(****************************************************************
NAME:			FB_Move
DATA:			2017.2.17
VERSION:		1.0.0
DESCRIPTION:	FB_Move
HISTORY:
				2017.2.17		NEW
				2018.1.9		ÐÂÔöBCGapMode
***************************************************************)
FUNCTION_BLOCK FB_Move
VAR_INPUT
	(*È«¾Ö*)
	Mode:DINT;
	PowerState:BOOL;
	CoupleState:DINT;
	(*BCGapMode*)
	BCLeftTopPosition:LREAL;
	BCLeftTopVelocity:LREAL;
	BCRightTopPosition:LREAL;
	BCRightTopVelocity:LREAL;
	BCLeftBottomPosition:LREAL;
	BCLeftBottomVelocity:LREAL;
	BCRightBottomPosition:LREAL;
	BCRightBottomVelocity:LREAL;
	BCGapMove:BOOL;
	BCGapReset:BOOL;
	BCGapMove_2:BOOL;
	BCGapReset_2:BOOL;
	(*GapMode*)
	GapPosition:LREAL;
	GapVelocity:LREAL;
	GapMove:BOOL;
	GapReset:BOOL;
	(*SingleCarrierMode*)
	TopPosition:LREAL;
	TopVelocity:LREAL;
	TopMove:BOOL;
	TopReset:BOOL;
	BottomPosition:LREAL;
	BottomVelocity:LREAL;
	BottomMove:BOOL;
	BottomReset:BOOL;
	(*TaperMode*)
	TaperPosition:LREAL;
	TaperVelocity:LREAL;
	TaperMove:BOOL;
	TaperStop:BOOL;
	TaperReset:BOOL;
	(**DebugMode*)
	LeftTopPosition:LREAL;
	LeftTopVelocity:LREAL;
	LeftTopMove:BOOL;
	LeftTopStop:BOOL;
	LeftTopReset:BOOL;
	RightTopPosition:LREAL;
	RightTopVelocity:LREAL;
	RightTopMove:BOOL;
	RightTopStop:BOOL;
	RightTopReset:BOOL;
	LeftBottomPosition:LREAL;
	LeftBottomVelocity:LREAL;
	LeftBottomMove:BOOL;
	LeftBottomStop:BOOL;
	LeftBottomReset:BOOL;
	RightBottomPosition:LREAL;
	RightBottomVelocity:LREAL;
	RightBottomMove:BOOL;
	RightBottomStop:BOOL;
	RightBottomReset:BOOL;
	PhaseUpperPosition:LREAL;
	PhaseUpperVelocity:LREAL;
	PhaseUpperMove:BOOL;
	PhaseUpperStop:BOOL;
	PhaseUpperReset:BOOL;
	PhaseLowerPosition:LREAL;
	PhaseLowerVelocity:LREAL;
	PhaseLowerMove:BOOL;
	PhaseLowerStop:BOOL;
	PhaseLowerReset:BOOL;
END_VAR
VAR_OUTPUT
	FbID:DINT:=1001;
	GapState:DINT;
	GapBusy:BOOL;
	GapDone:BOOL;
	GapMoving:BOOL;

	BCGapState:DINT;
	BCGapBusy:BOOL;
	BCGapDone:BOOL;

	TopState:DINT;
	TopBusy:BOOL;
	TopDone:BOOL;
	BottomState:DINT;
	BottomBusy:BOOL;
	BottomDone:BOOL;

	TaperState:DINT;
	TaperBusy:BOOL;
	TaperDone:BOOL;

	LeftTopState:DINT;
	LeftTopBusy:BOOL;
	LeftTopDone:BOOL;
	RightTopState:DINT;
	RightTopBusy:BOOL;
	RightTopDone:BOOL;
	LeftBottomState:DINT;
	LeftBottomBusy:BOOL;
	LeftBottomDone:BOOL;
	RightBottomState:DINT;
	RightBottomBusy:BOOL;
	RightBottomDone:BOOL;
	PhaseUpperState:DINT;
	PhaseUpperBusy:BOOL;
	PhaseUpperDone:BOOL;
	PhaseLowerState:DINT;
	PhaseLowerBusy:BOOL;
	PhaseLowerDone:BOOL;

	Error:BOOL;
	ErrorID:DINT;
	
	GapState_2:DINT;
	GapBusy_2:BOOL;
	GapDone_2:BOOL;

	BCGapState_2:DINT;
	BCGapBusy_2:BOOL;
	BCGapDone_2:BOOL;
END_VAR
VAR
	Top_MC_MoveAbsolute: MC_MoveAbsolute;
	Bottom_MC_MoveAbsolute: MC_MoveAbsolute;
	RightTopLin_MC_MoveAbsolute: MC_MoveAbsolute;
	RightBottomLin_MC_MoveAbsolute: MC_MoveAbsolute;
	PhaseUpperLin_MC_MoveAbsolute: MC_MoveAbsolute;
	PhaseLowerLin_MC_MoveAbsolute: MC_MoveAbsolute;
	fb_ton: TON;
	fb_ton1: TON;
	fb_ton2: TON;
	fb_ton_debug_1:TON;
	fb_ton_debug_2:TON;
	fb_ton_debug_3:TON;
	fb_ton_debug_4:TON;
	fb_ton_debug_5:TON;
	fb_ton_debug_6:TON;
	fb_ton_BC:TON;
	fb_ton_BC_2:TON;
END_VAR

IF PowerState=1 THEN
	IF Mode=1 AND CoupleState=1 THEN
		A_GapMove();
	ELSIF Mode=2 AND CoupleState=0 AND TopMove THEN
		A_TopMove();
	ELSIF Mode=2 AND CoupleState=0 AND BottomMove THEN
		A_BottomMove();
	ELSIF Mode=3 AND CoupleState=0 AND TaperMove THEN
		A_TaperMove();
	ELSIF Mode=4 AND CoupleState=0 AND LeftTopMove THEN
		A_LeftTopMove();
	ELSIF Mode=4 AND CoupleState=0 AND RightTopMove THEN
		A_RightTopMove();
	ELSIF Mode=4 AND CoupleState=0 AND LeftBottomMove THEN
		A_LeftBottomMove();
	ELSIF Mode=4 AND CoupleState=0 AND RightBottomMove THEN
		A_RightBottomMove();
	ELSIF Mode=4 AND CoupleState=0 AND PhaseUpperMove THEN
		A_PhaseUpperMove();
	ELSIF Mode=4 AND CoupleState=0 AND PhaseLowerMove THEN
		A_PhaseLowerMove();
	ELSIF Mode=5 AND CoupleState=0 AND BCGapMove THEN
		A_BCGapMove();
	ELSIF Mode=6 AND CoupleState=0 AND BCGapMove_2 THEN
		A_BCGapMove_2();
	END_IF
END_IF

ACTION A_BCGapMove:
IF BCGapMove THEN
	BCGapBusy:=TRUE;
	BCGapDone:=FALSE;
	fb_ton_BC(PT:=t#80s);(*2mm/s max spees,120mmÐÐ³Ì£¬60sÄÚ×ßÍê*)
	(*×îºóÔÙ¼ì²éÒ»±éñîºÏ£¬²¹³¥Ä£Ê½ÏÂ£¬²»ÄÜñîºÏ*)
	IF LeftTopLin.NcToPlc.CoupleState<>0 OR LeftBottomLin.NcToPlc.CoupleState<>0
				OR RightTopLin.NcToPlc.CoupleState<>0 OR RightBottomLin.NcToPlc.CoupleState<>0 THEN
				ErrorID:=1;
				GapState:=-100;
	END_IF
	A_MoveMC();
	IF  LeftTopLin.Status.Moving AND RightTopLin.Status.Moving
				 AND LeftBottomLin.Status.Moving AND RightBottomLin.Status.Moving THEN
		GapMoving:=TRUE;
	ELSE
		GapMoving:=FALSE;
	END_IF
	CASE BCGapState OF
		0:
			IF LeftTopLin.Status.Moving OR RightTopLin.Status.Moving
				 OR LeftBottomLin.Status.Moving OR RightBottomLin.Status.Moving THEN	(*ÖáÕýÔÚÔËÐÐ£¬Ñ­»·¸Ã²½µÈ´ý*)
				BCGapState:=88;
			//ELSIF Top_MC_MoveAbsolute.Error OR Bottom_MC_MoveAbsolute.Error OR
			//		RightTopLin_MC_MoveAbsolute.Error OR RightBottomLin_MC_MoveAbsolute.Error THEN	(*¼ì²éMC Error*)
			//	ErrorID:=2;
			//	BCGapState:=99;
			(*ELSIF ABS(Pos_LeftTopLin-GapPosition/2)<0.002 AND  ABS(Pos_LeftBottomLin-GapPosition)<0.002 THEN	(*Ä¿±êÎ»ÖÃÓëµ±Ç°Î»ÖÃÒ»Ñù£¬²»¶¯*)
				GapState:=88;*)
			ELSIF leftTopLin.Status.NotMoving AND  leftBottomLin.Status.NotMoving
				 AND RightTopLin.Status.NotMoving AND RightBottomLin.Status.NotMoving THEN	(*Öá¶¼´¦ÓÚÍ£Ö¹×´Ì¬Ê±£¬×ªÏÂÒ»²½*)
				BCGapState:=1;
			END_IF
		1:
			Top_MC_MoveAbsolute.Position:=BCLeftTopPosition;
			Top_MC_MoveAbsolute.Velocity:=BCLeftTopVelocity;
			Bottom_MC_MoveAbsolute.Position:=BCLeftBottomPosition;
			Bottom_MC_MoveAbsolute.Velocity:=BCLeftBottomVelocity;
			RightTopLin_MC_MoveAbsolute.Position:=BCRightTopPosition;
			RightTopLin_MC_MoveAbsolute.Velocity:=BCRightTopVelocity;
			RightBottomLin_MC_MoveAbsolute.Position:=BCRightBottomPosition;
			RightBottomLin_MC_MoveAbsolute.Velocity:=BCRightBottomVelocity;
			Top_MC_MoveAbsolute.Execute:=TRUE;
			Bottom_MC_MoveAbsolute.Execute:=TRUE;
			RightTopLin_MC_MoveAbsolute.Execute:=TRUE;
			RightBottomLin_MC_MoveAbsolute.Execute:=TRUE;
			fb_ton_BC.IN:=TRUE;
			BCGapState:=2;
		2:
			IF NOT Top_MC_MoveAbsolute.Done OR NOT  Bottom_MC_MoveAbsolute.Done
					OR NOT RightTopLin_MC_MoveAbsolute.Done OR NOT RightBottomLin_MC_MoveAbsolute.Done THEN		(*ÔË¶¯ÖÐ£¬¼ì²éDoneÐÅºÅ£¬Ã»ÓÐÔòÑ­»·*)
				BCGapState:=2;
			ELSIF Top_MC_MoveAbsolute.Done  AND  Bottom_MC_MoveAbsolute.Done AND RightTopLin_MC_MoveAbsolute.Done AND RightBottomLin_MC_MoveAbsolute.Done THEN		(*ÔË¶¯Íê³É£¬×ªÏÂÒ»²½*)
				BCGapState:=88;
			END_IF
		88:
			BCGapMove:=FALSE;
			BCGapState:=0;
			BCGapBusy:=FALSE;
			BCGapDone:=TRUE;
			Error:=FALSE;
			ErrorID:=0;
			Top_MC_MoveAbsolute.Execute:=FALSE;
			Bottom_MC_MoveAbsolute.Execute:=FALSE;
			RightTopLin_MC_MoveAbsolute.Execute:=FALSE;
			RightBottomLin_MC_MoveAbsolute.Execute:=FALSE;
			fb_ton_BC.IN:=FALSE;
		89:
			BCGapMove:=FALSE;
			BCGapState:=0;
			BCGapBusy:=FALSE;
			BCGapDone:=FALSE;
			Error:=FALSE;
			ErrorID:=0;
			Top_MC_MoveAbsolute.Execute:=FALSE;
			Bottom_MC_MoveAbsolute.Execute:=FALSE;
			RightTopLin_MC_MoveAbsolute.Execute:=FALSE;
			RightBottomLin_MC_MoveAbsolute.Execute:=FALSE;
			fb_ton_BC.IN:=FALSE;
		99:
			BCGapMove:=FALSE;
			BCGapState:=99;
			BCGapBusy:=FALSE;
			BCGapDone:=FALSE;
			Error:=TRUE;
			Top_MC_MoveAbsolute.Execute:=FALSE;
			Bottom_MC_MoveAbsolute.Execute:=FALSE;
			RightTopLin_MC_MoveAbsolute.Execute:=FALSE;
			RightBottomLin_MC_MoveAbsolute.Execute:=FALSE;
			fb_ton_BC.IN:=FALSE;
		-100:
			FB_PlcEmergencyStop();
			BCGapMove:=FALSE;
			BCGapState:=-100;
			BCGapBusy:=FALSE;
			BCGapDone:=FALSE;
			Error:=TRUE;
			Top_MC_MoveAbsolute.Execute:=FALSE;
			Bottom_MC_MoveAbsolute.Execute:=FALSE;
			RightTopLin_MC_MoveAbsolute.Execute:=FALSE;
			RightBottomLin_MC_MoveAbsolute.Execute:=FALSE;
			fb_ton_BC.IN:=FALSE;
	END_CASE

	IF BCGapReset THEN
		BCGapReset:=FALSE;
		BCGapMove:=FALSE;
		BCGapState:=0;
		BCGapBusy:=FALSE;
		BCGapDone:=FALSE;
		Error:=FALSE;
		ErrorID:=0;
		Top_MC_MoveAbsolute.Execute:=FALSE;
		Bottom_MC_MoveAbsolute.Execute:=FALSE;
		RightTopLin_MC_MoveAbsolute.Execute:=FALSE;
		RightBottomLin_MC_MoveAbsolute.Execute:=FALSE;
		fb_ton_BC.IN:=FALSE;
	END_IF
END_IF
END_ACTION

ACTION A_BCGapMove_2:
IF BCGapMove_2 THEN
BCGapBusy_2:=TRUE;
BCGapDone_2:=FALSE;
fb_ton_BC_2(PT:=T#80S);(*2mm/s max spees,120mmÐÐ³Ì£¬60sÄÚ×ßÍê*)
(*×îºóÔÙ¼ì²éÒ»±éñîºÏ£¬²¹³¥Ä£Ê½ÏÂ£¬²»ÄÜñîºÏ*)
IF LeftTopLin.NcToPlc.CoupleState<>0 OR LeftBottomLin.NcToPlc.CoupleState<>0
			OR RightTopLin.NcToPlc.CoupleState<>0 OR RightBottomLin.NcToPlc.CoupleState<>0 THEN
			ErrorID:=1;
			GapState:=-100;
END_IF
A_MoveMC();
CASE BCGapState_2 OF
	0:
		IF LeftTopLin.Status.Moving OR RightTopLin.Status.Moving
			 OR LeftBottomLin.Status.Moving OR RightBottomLin.Status.Moving THEN	(*ÖáÕýÔÚÔËÐÐ£¬Ñ­»·¸Ã²½µÈ´ý*)
			BCGapState_2:=88;
		//ELSIF Top_MC_MoveAbsolute.Error OR Bottom_MC_MoveAbsolute.Error OR
		//		RightTopLin_MC_MoveAbsolute.Error OR RightBottomLin_MC_MoveAbsolute.Error THEN	(*¼ì²éMC Error*)
		//	ErrorID:=2;
		//	BCGapState_2:=99;
		(*ELSIF ABS(Pos_LeftTopLin-GapPosition/2)<0.002 AND  ABS(Pos_LeftBottomLin-GapPosition)<0.002 THEN	(*Ä¿±êÎ»ÖÃÓëµ±Ç°Î»ÖÃÒ»Ñù£¬²»¶¯*)
			GapState:=88;*)
		ELSIF leftTopLin.Status.NotMoving AND  leftBottomLin.Status.NotMoving
			 AND RightTopLin.Status.NotMoving AND RightBottomLin.Status.NotMoving THEN	(*Öá¶¼´¦ÓÚÍ£Ö¹×´Ì¬Ê±£¬×ªÏÂÒ»²½*)
			BCGapState_2:=1;
		END_IF
	1:
		Top_MC_MoveAbsolute.Position:=BCLeftTopPosition;
		Top_MC_MoveAbsolute.Velocity:=BCLeftTopVelocity;
		Bottom_MC_MoveAbsolute.Position:=BCLeftBottomPosition;
		Bottom_MC_MoveAbsolute.Velocity:=BCLeftBottomVelocity;
		RightTopLin_MC_MoveAbsolute.Position:=BCRightTopPosition;
		RightTopLin_MC_MoveAbsolute.Velocity:=BCRightTopVelocity;
		RightBottomLin_MC_MoveAbsolute.Position:=BCRightBottomPosition;
		RightBottomLin_MC_MoveAbsolute.Velocity:=BCRightBottomVelocity;
		Top_MC_MoveAbsolute.Execute:=TRUE;
		Bottom_MC_MoveAbsolute.Execute:=TRUE;
		RightTopLin_MC_MoveAbsolute.Execute:=TRUE;
		RightBottomLin_MC_MoveAbsolute.Execute:=TRUE;
		fb_ton_BC_2.IN:=TRUE;
		BCGapState_2:=2;
	2:
		IF NOT Top_MC_MoveAbsolute.Done OR NOT  Bottom_MC_MoveAbsolute.Done
				OR NOT RightTopLin_MC_MoveAbsolute.Done OR NOT RightBottomLin_MC_MoveAbsolute.Done THEN		(*ÔË¶¯ÖÐ£¬¼ì²éDoneÐÅºÅ£¬Ã»ÓÐÔòÑ­»·*)
			BCGapState_2:=2;
		ELSIF Top_MC_MoveAbsolute.Done  AND  Bottom_MC_MoveAbsolute.Done AND RightTopLin_MC_MoveAbsolute.Done AND RightBottomLin_MC_MoveAbsolute.Done THEN		(*ÔË¶¯Íê³É£¬×ªÏÂÒ»²½*)
			BCGapState_2:=88;
		END_IF
		(*½ÓÊÕµ½stopÐÅºÅÊ±£¬reset×´Ì¬*)
		IF BCGapReset_2 THEN
			BCGapState_2:=89;
		END_IF

	88:
		BCGapMove_2:=FALSE;
		BCGapState_2:=0;
		BCGapBusy_2:=FALSE;
		BCGapDone_2:=TRUE;
		Error:=FALSE;
		ErrorID:=0;
		Top_MC_MoveAbsolute.Execute:=FALSE;
		Bottom_MC_MoveAbsolute.Execute:=FALSE;
		RightTopLin_MC_MoveAbsolute.Execute:=FALSE;
		RightBottomLin_MC_MoveAbsolute.Execute:=FALSE;
		fb_ton_BC_2.IN:=FALSE;
	89:
		BCGapMove_2:=FALSE;
		BCGapState_2:=0;
		BCGapBusy_2:=FALSE;
		BCGapDone_2:=FALSE;
		Error:=FALSE;
		ErrorID:=0;
		Top_MC_MoveAbsolute.Execute:=FALSE;
		Bottom_MC_MoveAbsolute.Execute:=FALSE;
		RightTopLin_MC_MoveAbsolute.Execute:=FALSE;
		RightBottomLin_MC_MoveAbsolute.Execute:=FALSE;
		fb_ton_BC_2.IN:=FALSE;
	99:
		BCGapMove_2:=FALSE;
		BCGapState_2:=99;
		BCGapBusy_2:=FALSE;
		BCGapDone_2:=FALSE;
		Error:=TRUE;
		Top_MC_MoveAbsolute.Execute:=FALSE;
		Bottom_MC_MoveAbsolute.Execute:=FALSE;
		RightTopLin_MC_MoveAbsolute.Execute:=FALSE;
		RightBottomLin_MC_MoveAbsolute.Execute:=FALSE;
		fb_ton_BC_2.IN:=FALSE;
	-100:
		FB_PlcEmergencyStop();
		BCGapMove_2:=FALSE;
		BCGapState_2:=-100;
		BCGapBusy_2:=FALSE;
		BCGapDone_2:=FALSE;
		Error:=TRUE;
		Top_MC_MoveAbsolute.Execute:=FALSE;
		Bottom_MC_MoveAbsolute.Execute:=FALSE;
		RightTopLin_MC_MoveAbsolute.Execute:=FALSE;
		RightBottomLin_MC_MoveAbsolute.Execute:=FALSE;
		fb_ton_BC_2.IN:=FALSE;
END_CASE
END_IF
END_ACTION

ACTION A_BottomMove:
IF BottomMove THEN
BottomBusy:=TRUE;
BottomDone:=FALSE;
fb_ton2(PT:=t#80s);(*2mm/s max spees,120mmÐÐ³Ì£¬60sÄÚ×ßÍê*)
A_MoveMC();
CASE BottomState OF

	0:
		IF LeftTopLin.Status.Moving OR RightTopLin.Status.Moving
			 OR LeftBottomLin.Status.Moving OR RightBottomLin.Status.Moving THEN	(*ÖáÕýÔÚÔËÐÐ£¬Ñ­»·¸Ã²½µÈ´ý*)
			TopState:=88;
		//ELSIF  Bottom_MC_MoveAbsolute.Error OR RightBottomLin_MC_MoveAbsolute.Error THEN		(*¼ì²éMC Error*)
		//	ErrorID:=2;
		//	BottomState:=99;
		ELSIF leftTopLin.Status.NotMoving AND  leftBottomLin.Status.NotMoving
			 AND RightTopLin.Status.NotMoving AND RightBottomLin.Status.NotMoving THEN	(*Öá¶¼´¦ÓÚÍ£Ö¹×´Ì¬Ê±£¬×ªÏÂÒ»²½*)
			BottomState:=1;
		END_IF
	1:
		Bottom_MC_MoveAbsolute.Position:=BottomPosition;
		Bottom_MC_MoveAbsolute.Velocity:=BottomVelocity;
		Bottom_MC_MoveAbsolute.Execute:=TRUE;
		RightBottomLin_MC_MoveAbsolute.Position:=BottomPosition;
		RightBottomLin_MC_MoveAbsolute.Velocity:=BottomVelocity;
		RightBottomLin_MC_MoveAbsolute.Execute:=TRUE;
		fb_ton2.IN:=TRUE;
		BottomState:=2;
	2:
		IF leftTopLin.Status.Moving OR RightTopLin.Status.Moving THEN	(*ÉÏÁº¶¯,ESTOP*)
			ErrorID:=3;
			BottomState:=-100;
		ELSIF  (LeftBottomLin.Status.Moving AND  RightBottomLin.Status.NotMoving)
				OR (RightBottomLin.Status.Moving AND  LeftBottomLin.Status.NotMoving) THEN
			//ErrorID:=4;
			//BottomState:=-100;
		ELSIF NOT Bottom_MC_MoveAbsolute.Done THEN		(*ÔË¶¯ÖÐ£¬¼ì²éDoneÐÅºÅ£¬Ã»ÓÐÔòÑ­»·£¬³¬Ê±±¨´í*)
			BottomState:=2;
		ELSIF Bottom_MC_MoveAbsolute.Done THEN		(*ÔË¶¯Íê³É£¬×ªÏÂÒ»²½*)
				BottomState:=88;
		END_IF
		(*½ÓÊÕµ½stopÐÅºÅÊ±£¬reset×´Ì¬*)
		IF BottomReset THEN
			BottomState:=89;
		END_IF

	88:
		BottomMove:=FALSE;
		BottomState:=0;
		BottomBusy:=FALSE;
		BottomDone:=TRUE;
		Error:=FALSE;
		ErrorID:=0;
		Bottom_MC_MoveAbsolute.Execute:=FALSE;
		RightBottomLin_MC_MoveAbsolute.Execute:=FALSE;
		fb_ton2.IN:=FALSE;
	89:
		BottomMove:=FALSE;
		BottomState:=0;
		BottomBusy:=FALSE;
		BottomDone:=FALSE;
		Error:=FALSE;
		ErrorID:=0;
		Bottom_MC_MoveAbsolute.Execute:=FALSE;
		RightBottomLin_MC_MoveAbsolute.Execute:=FALSE;
		fb_ton2.IN:=FALSE;
	99:
		BottomMove:=FALSE;
		BottomState:=99;
		BottomBusy:=FALSE;
		BottomDone:=FALSE;
		Error:=TRUE;
		Bottom_MC_MoveAbsolute.Execute:=FALSE;
		RightBottomLin_MC_MoveAbsolute.Execute:=FALSE;
		fb_ton2.IN:=FALSE;
	-100:
		FB_PlcEmergencyStop();
		BottomMove:=FALSE;
		BottomState:=-100;
		BottomBusy:=FALSE;
		BottomDone:=FALSE;
		Error:=TRUE;
		Bottom_MC_MoveAbsolute.Execute:=FALSE;
		RightBottomLin_MC_MoveAbsolute.Execute:=FALSE;
		fb_ton2.IN:=FALSE;
END_CASE
END_IF
END_ACTION

ACTION A_GapMove:
IF GapMove THEN
GapBusy:=TRUE;
GapDone:=FALSE;
fb_ton(PT:=t#80s);(*2mm/s max spees,120mmÐÐ³Ì£¬60sÄÚ×ßÍê*)
(*×îºóÔÙ¼ì²éÒ»±éñîºÏ*)
IF LeftTopLin.NcToPlc.CoupleState<>1 OR LeftBottomLin.NcToPlc.CoupleState<>1
			OR RightTopLin.NcToPlc.CoupleState<>3 OR RightBottomLin.NcToPlc.CoupleState<>3 THEN
			ErrorID:=1;
			GapState:=-100;
END_IF
A_MoveMC();
CASE GapState OF

	0:
		IF LeftTopLin.Status.Moving OR RightTopLin.Status.Moving
			 OR LeftBottomLin.Status.Moving OR RightBottomLin.Status.Moving THEN	(*ÖáÕýÔÚÔËÐÐ£¬Ñ­»·¸Ã²½µÈ´ý*)
			GapState:=88;
		//ELSIF Top_MC_MoveAbsolute.Error OR Bottom_MC_MoveAbsolute.Error THEN		(*¼ì²éMC Error*)
		//	ErrorID:=2;
		//	GapState:=99;
		ELSIF ABS(Pos_LeftTopLin-GapPosition/2)<0.002 AND  ABS(Pos_LeftBottomLin-GapPosition)<0.002 THEN	(*Ä¿±êÎ»ÖÃÓëµ±Ç°Î»ÖÃÒ»Ñù£¬²»¶¯*)
			GapState:=88;
		ELSIF leftTopLin.Status.NotMoving AND  leftBottomLin.Status.NotMoving
			 AND RightTopLin.Status.NotMoving AND RightBottomLin.Status.NotMoving THEN	(*Öá¶¼´¦ÓÚÍ£Ö¹×´Ì¬Ê±£¬×ªÏÂÒ»²½*)
			GapState:=1;
		END_IF
	1:
		Top_MC_MoveAbsolute.Position:=GapPosition/2;
		Top_MC_MoveAbsolute.Velocity:=GapVelocity/2;
		Bottom_MC_MoveAbsolute.Position:=GapPosition/2;
		Bottom_MC_MoveAbsolute.Velocity:=GapVelocity/2;
		Top_MC_MoveAbsolute.Execute:=TRUE;
		Bottom_MC_MoveAbsolute.Execute:=TRUE;
		fb_ton.IN:=TRUE;
		GapState:=2;
	2:
		(*IF leftTopLin.Status.Moving AND   leftBottomLin.Status.NotMoving THEN (*ÉÏÏÂÁº²»Í¬Ê±¶¯*)
			ErrorID:=3;
			GapState:=-100;
		ELSIF RightTopLin.Status.NotMoving AND RightBottomLin.Status.Moving THEN (*ÉÏÏÂÁº²»Í¬Ê±¶¯*)
			ErrorID:=4;
			GapState:=-100;
		*)
		IF  (LeftTopLin.Status.Moving AND  RightTopLin.Status.NotMoving)
			OR  (LeftTopLin.Status.Moving AND LeftBottomLin.Status.NotMoving)
			OR (LeftTopLin.Status.Moving AND  RightBottomLin.Status.NotMoving)
				OR (RightTopLin.Status.Moving AND  LeftTopLin.Status.NotMoving)
				OR (RightTopLin.Status.Moving AND  LeftBottomLin.Status.NotMoving)
				OR (RightTopLin.Status.Moving AND  RightBottomLin.Status.NotMoving)
					OR (LeftBottomLin.Status.Moving AND  LeftTopLin.Status.NotMoving)
					OR (LeftBottomLin.Status.Moving AND  RightTopLin.Status.NotMoving)
					OR (LeftBottomLin.Status.Moving AND  RightBottomLin.Status.NotMoving)
						OR (RightBottomLin.Status.Moving AND  LeftTopLin.Status.NotMoving)
						OR (RightBottomLin.Status.Moving AND  RightTopLin.Status.NotMoving)
						OR (RightBottomLin.Status.Moving AND  LeftBottomLin.Status.NotMoving) THEN			(*Ò»Öá¶¯£¬ÆäËüÖá²»¶¯£¬½ô¼±×´Ì¬*)
			ErrorID:=5;
			GapState:=-100;
		ELSIF NOT Top_MC_MoveAbsolute.Done OR NOT  Bottom_MC_MoveAbsolute.Done THEN		(*ÔË¶¯ÖÐ£¬¼ì²éDoneÐÅºÅ£¬Ã»ÓÐÔòÑ­»·£¬³¬Ê±±¨´í*)
			(*IF NOT  fb_ton.Q THEN
				GapState:=2;
			ELSE
				ErrorID:=5;
				GapState:=-100;
			END_IF*)
			GapState:=2;
		ELSIF Top_MC_MoveAbsolute.Done  AND  Bottom_MC_MoveAbsolute.Done THEN		(*ÔË¶¯Íê³É£¬×ªÏÂÒ»²½*)
				GapState:=88;
		END_IF
		(*½ÓÊÕµ½stopÐÅºÅÊ±£¬reset×´Ì¬*)
		IF GapReset THEN
			GapState:=89;
		END_IF

	88:
		GapMove:=FALSE;
		GapState:=0;
		GapBusy:=FALSE;
		GapDone:=TRUE;
		Error:=FALSE;
		ErrorID:=0;
		Top_MC_MoveAbsolute.Execute:=FALSE;
		Bottom_MC_MoveAbsolute.Execute:=FALSE;
		fb_ton.IN:=FALSE;
	89:
		GapMove:=FALSE;
		GapState:=0;
		GapBusy:=FALSE;
		GapDone:=FALSE;
		Error:=FALSE;
		ErrorID:=0;
		Top_MC_MoveAbsolute.Execute:=FALSE;
		Bottom_MC_MoveAbsolute.Execute:=FALSE;
		fb_ton.IN:=FALSE;
	99:
		GapMove:=FALSE;
		GapState:=99;
		GapBusy:=FALSE;
		GapDone:=FALSE;
		Error:=TRUE;
		Top_MC_MoveAbsolute.Execute:=FALSE;
		Bottom_MC_MoveAbsolute.Execute:=FALSE;
		fb_ton.IN:=FALSE;
	-100:
		FB_PlcEmergencyStop();
		GapMove:=FALSE;
		GapState:=-100;
		GapBusy:=FALSE;
		GapDone:=FALSE;
		Error:=TRUE;
		Top_MC_MoveAbsolute.Execute:=FALSE;
		Bottom_MC_MoveAbsolute.Execute:=FALSE;
		fb_ton.IN:=FALSE;
END_CASE
END_IF
END_ACTION

ACTION A_LeftBottomMove:
IF LeftBottomMove THEN
LeftBottomBusy:=TRUE;
LeftBottomDone:=FALSE;
fb_ton_debug_3(PT:=t#10s);
(*×îºóÔÙ¼ì²éÒ»±éñîºÏ£¬²»ñîºÏÎªÕýÈ·×´Ì¬*)
IF LeftTopLin.NcToPlc.CoupleState<>0 OR LeftBottomLin.NcToPlc.CoupleState<>0
			OR RightTopLin.NcToPlc.CoupleState<>0 OR RightBottomLin.NcToPlc.CoupleState<>0 THEN
			ErrorID:=1;
			LeftBottomState:=-100;
END_IF
A_MoveMC();
CASE LeftBottomState OF
	0:
		//IF Top_MC_MoveAbsolute.Error OR Bottom_MC_MoveAbsolute.Error
		//	OR RightTopLin_MC_MoveAbsolute.Error OR RightBottomLin_MC_MoveAbsolute.Error THEN		(*¼ì²éMC Error*)
		//	ErrorID:=2;
		//	LeftBottomState:=99;
		IF leftTopLin.Status.NotMoving AND  leftBottomLin.Status.NotMoving
			 AND RightTopLin.Status.NotMoving AND RightBottomLin.Status.NotMoving THEN	(*Öá¶¼´¦ÓÚÍ£Ö¹×´Ì¬Ê±£¬×ªÏÂÒ»²½*)
			LeftBottomState:=1;
		END_IF
	1:
		Bottom_MC_MoveAbsolute.Position:=LeftBottomPosition;
		Bottom_MC_MoveAbsolute.Velocity:=LeftBottomVelocity;
		Bottom_MC_MoveAbsolute.Execute:=TRUE;
		fb_ton_debug_3.IN:=TRUE;
		LeftBottomState:=2;
	2:
		IF LeftTopLin.Status.Moving OR RightTopLin.Status.Moving OR RightBottomLin.Status.Moving THEN	(*³ýÁËÔË¶¯Öá¶¯£¬ÆäÓàÖáÓÐ¶¯£¬´íÎó*)
			ErrorID:=3;
			LeftBottomState:=-100;
		ELSIF NOT Bottom_MC_MoveAbsolute.Done THEN		(*ÔË¶¯ÖÐ£¬¼ì²éDoneÐÅºÅ£¬Ã»ÓÐÔòÑ­»·£¬³¬Ê±±¨´í*)
			(*IF NOT  fb_ton.Q THEN
				LeftBottomState:=2;
			ELSE
				ErrorID:=5;
				LeftBottomState:=-100;
			END_IF*)
			LeftBottomState:=2;
		ELSIF Bottom_MC_MoveAbsolute.Done THEN		(*ÔË¶¯Íê³É£¬×ªÏÂÒ»²½*)
				LeftBottomState:=88;
		END_IF
		(*½ÓÊÕµ½stopÐÅºÅÊ±£¬reset×´Ì¬*)
		IF LeftBottomReset THEN
			LeftBottomState:=89;
		END_IF

	88:
		LeftBottomMove:=FALSE;
		LeftBottomState:=0;
		LeftBottomBusy:=FALSE;
		LeftBottomDone:=TRUE;
		Error:=FALSE;
		ErrorID:=0;
		Bottom_MC_MoveAbsolute.Execute:=FALSE;
		fb_ton_debug_3.IN:=FALSE;
	89:
		LeftBottomMove:=FALSE;
		LeftBottomState:=0;
		LeftBottomBusy:=FALSE;
		LeftBottomDone:=FALSE;
		Error:=FALSE;
		ErrorID:=0;
		Bottom_MC_MoveAbsolute.Execute:=FALSE;
		fb_ton_debug_3.IN:=FALSE;
	99:
		LeftBottomMove:=FALSE;
		LeftBottomState:=99;
		LeftBottomBusy:=FALSE;
		LeftBottomDone:=FALSE;
		Error:=TRUE;
		Bottom_MC_MoveAbsolute.Execute:=FALSE;
		fb_ton_debug_3.IN:=FALSE;
	-100:
		FB_PlcEmergencyStop();
		LeftBottomMove:=FALSE;
		LeftBottomState:=-100;
		LeftBottomBusy:=FALSE;
		LeftBottomDone:=FALSE;
		Error:=TRUE;
		Bottom_MC_MoveAbsolute.Execute:=FALSE;
		fb_ton_debug_3.IN:=FALSE;
END_CASE
END_IF
END_ACTION

ACTION A_LeftTopMove:
IF LeftTopMove THEN
LeftTopBusy:=TRUE;
LeftTopDone:=FALSE;
fb_ton_debug_1(PT:=t#10s);
(*×îºóÔÙ¼ì²éÒ»±éñîºÏ£¬²»ñîºÏÎªÕýÈ·×´Ì¬*)
IF LeftTopLin.NcToPlc.CoupleState<>0 OR LeftBottomLin.NcToPlc.CoupleState<>0
			OR RightTopLin.NcToPlc.CoupleState<>0 OR RightBottomLin.NcToPlc.CoupleState<>0 THEN
			ErrorID:=1;
			LeftTopState:=-100;
END_IF
A_MoveMC();
CASE LeftTopState OF
	0:
		//IF Top_MC_MoveAbsolute.Error OR Bottom_MC_MoveAbsolute.Error
		//	OR RightTopLin_MC_MoveAbsolute.Error OR RightBottomLin_MC_MoveAbsolute.Error THEN		(*¼ì²éMC Error*)
		//	ErrorID:=2;
		//	LeftTopState:=99;
		IF leftTopLin.Status.NotMoving AND  leftBottomLin.Status.NotMoving
			 AND RightTopLin.Status.NotMoving AND RightBottomLin.Status.NotMoving THEN	(*Öá¶¼´¦ÓÚÍ£Ö¹×´Ì¬Ê±£¬×ªÏÂÒ»²½*)
			LeftTopState:=1;
		END_IF
	1:
		Top_MC_MoveAbsolute.Position:=LeftTopPosition;
		Top_MC_MoveAbsolute.Velocity:=LeftTopVelocity;
		Top_MC_MoveAbsolute.Execute:=TRUE;
		fb_ton_debug_1.IN:=TRUE;
		LeftTopState:=2;
	2:
		IF RightTopLin.Status.Moving OR LeftBottomLin.Status.Moving OR RightBottomLin.Status.Moving THEN	(*³ýÁËÔË¶¯Öá¶¯£¬ÆäÓàÖáÓÐ¶¯£¬´íÎó*)
			ErrorID:=3;
			LeftTopState:=-100;
		ELSIF NOT Top_MC_MoveAbsolute.Done THEN		(*ÔË¶¯ÖÐ£¬¼ì²éDoneÐÅºÅ£¬Ã»ÓÐÔòÑ­»·£¬³¬Ê±±¨´í*)
			(*IF NOT  fb_ton.Q THEN
				LeftTopState:=2;
			ELSE
				ErrorID:=5;
				LeftTopState:=-100;
			END_IF*)
			LeftTopState:=2;
		ELSIF Top_MC_MoveAbsolute.Done THEN		(*ÔË¶¯Íê³É£¬×ªÏÂÒ»²½*)
				LeftTopState:=88;
		END_IF
		(*½ÓÊÕµ½stopÐÅºÅÊ±£¬reset×´Ì¬*)
		IF LeftTopReset THEN
			LeftTopState:=89;
		END_IF

	88:
		LeftTopMove:=FALSE;
		LeftTopState:=0;
		LeftTopBusy:=FALSE;
		LeftTopDone:=TRUE;
		Error:=FALSE;
		ErrorID:=0;
		Top_MC_MoveAbsolute.Execute:=FALSE;
		fb_ton_debug_1.IN:=FALSE;
	89:
		LeftTopMove:=FALSE;
		LeftTopState:=0;
		LeftTopBusy:=FALSE;
		LeftTopDone:=FALSE;
		Error:=FALSE;
		ErrorID:=0;
		Top_MC_MoveAbsolute.Execute:=FALSE;
		fb_ton_debug_1.IN:=FALSE;
	99:
		LeftTopMove:=FALSE;
		LeftTopState:=99;
		LeftTopBusy:=FALSE;
		LeftTopDone:=FALSE;
		Error:=TRUE;
		Top_MC_MoveAbsolute.Execute:=FALSE;
		fb_ton_debug_1.IN:=FALSE;
	-100:
		FB_PlcEmergencyStop();
		LeftTopMove:=FALSE;
		LeftTopState:=-100;
		LeftTopBusy:=FALSE;
		LeftTopDone:=FALSE;
		Error:=TRUE;
		Top_MC_MoveAbsolute.Execute:=FALSE;
		fb_ton_debug_1.IN:=FALSE;
END_CASE
END_IF
END_ACTION

ACTION A_MoveMC:
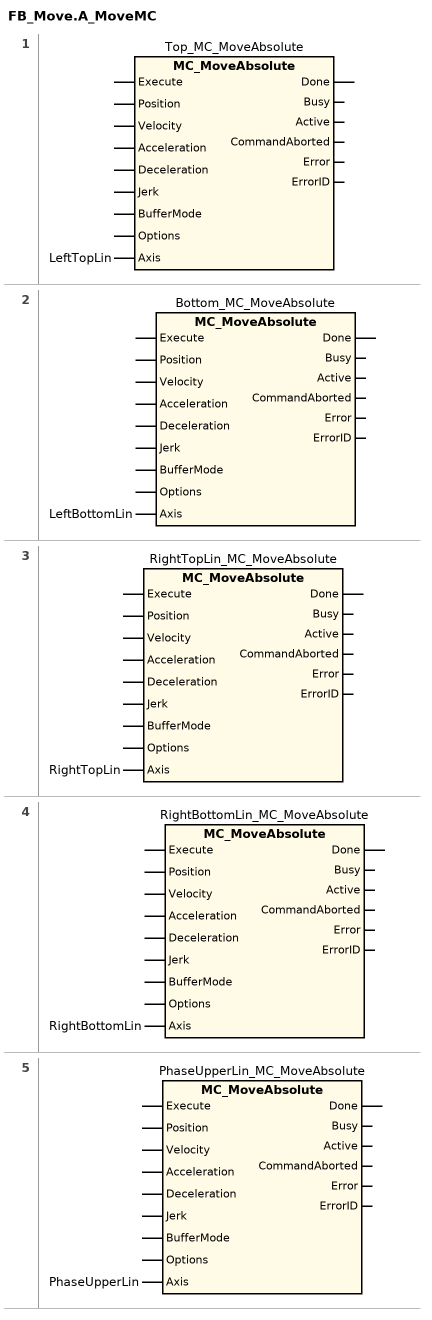
// NETWORK 1
Top_MC_MoveAbsolute(Axis := LeftTopLin); // MC_MoveAbsolute

// NETWORK 2
Bottom_MC_MoveAbsolute(Axis := LeftBottomLin); // MC_MoveAbsolute

// NETWORK 3
RightTopLin_MC_MoveAbsolute(Axis := RightTopLin); // MC_MoveAbsolute

// NETWORK 4
RightBottomLin_MC_MoveAbsolute(Axis := RightBottomLin); // MC_MoveAbsolute

// NETWORK 5
PhaseUpperLin_MC_MoveAbsolute(Axis := PhaseUpperLin); // MC_MoveAbsolute

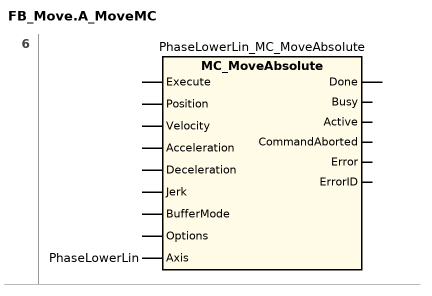
// NETWORK 6
PhaseLowerLin_MC_MoveAbsolute(Axis := PhaseLowerLin); // MC_MoveAbsolute
END_ACTION

ACTION A_PhaseLowerMove:
IF PhaseLowerMove THEN
PhaseLowerBusy:=TRUE;
PhaseLowerDone:=FALSE;
fb_ton_debug_6(PT:=T#10S);
A_MoveMC();
CASE PhaseLowerState OF
	0:
		//IF PhaseLowerLin_MC_MoveAbsolute.Error THEN
		//	ErrorID:=2;
		//	PhaseLowerState:=99;
		IF PhaseLowerLin.Status.NotMoving THEN	(*Öá¶¼´¦ÓÚÍ£Ö¹×´Ì¬Ê±£¬×ªÏÂÒ»²½*)
			PhaseLowerState:=1;
		END_IF
	1:
		PhaseLowerLin_MC_MoveAbsolute.Position:=PhaseLowerPosition;
		PhaseLowerLin_MC_MoveAbsolute.Velocity:=PhaseLowerVelocity;
		PhaseLowerLin_MC_MoveAbsolute.Execute:=TRUE;
		fb_ton_debug_6.IN:=TRUE;
		PhaseLowerState:=2;
	2:
		IF NOT PhaseLowerLin_MC_MoveAbsolute.Done THEN
			PhaseLowerState:=2;
		ELSIF PhaseLowerLin_MC_MoveAbsolute.Done THEN
				PhaseLowerState:=88;
		END_IF
		IF PhaseLowerReset THEN
			PhaseLowerState:=89;
		END_IF

	88:
		PhaseLowerMove:=FALSE;
		PhaseLowerState:=0;
		PhaseLowerBusy:=FALSE;
		PhaseLowerDone:=TRUE;
		Error:=FALSE;
		ErrorID:=0;
		PhaseLowerLin_MC_MoveAbsolute.Execute:=FALSE;
		fb_ton_debug_6.IN:=FALSE;
	89:
		PhaseLowerMove:=FALSE;
		PhaseLowerState:=0;
		PhaseLowerBusy:=FALSE;
		PhaseLowerDone:=FALSE;
		Error:=FALSE;
		ErrorID:=0;
		PhaseLowerLin_MC_MoveAbsolute.Execute:=FALSE;
		fb_ton_debug_6.IN:=FALSE;
	99:
		PhaseLowerMove:=FALSE;
		PhaseLowerState:=99;
		PhaseLowerBusy:=FALSE;
		PhaseLowerDone:=FALSE;
		Error:=TRUE;
		PhaseLowerLin_MC_MoveAbsolute.Execute:=FALSE;
		fb_ton_debug_6.IN:=FALSE;
	-100:
		FB_PlcEmergencyStop();
		PhaseLowerMove:=FALSE;
		PhaseLowerState:=-100;
		PhaseLowerBusy:=FALSE;
		PhaseLowerDone:=FALSE;
		Error:=TRUE;
		PhaseLowerLin_MC_MoveAbsolute.Execute:=FALSE;
		fb_ton_debug_6.IN:=FALSE;
END_CASE
END_IF
END_ACTION

ACTION A_PhaseUpperMove:
IF PhaseUpperMove THEN
PhaseUpperBusy:=TRUE;
PhaseUpperDone:=FALSE;
fb_ton_debug_5(PT:=T#10S);
A_MoveMC();
CASE PhaseUpperState OF
	0:
		//IF PhaseUpperLin_MC_MoveAbsolute.Error THEN
		//	ErrorID:=2;
		//	PhaseUpperState:=99;
		IF PhaseUpperLin.Status.NotMoving THEN	(*Öá¶¼´¦ÓÚÍ£Ö¹×´Ì¬Ê±£¬×ªÏÂÒ»²½*)
			PhaseUpperState:=1;
		END_IF
	1:
		PhaseUpperLin_MC_MoveAbsolute.Position:=PhaseUpperPosition;
		PhaseUpperLin_MC_MoveAbsolute.Velocity:=PhaseUpperVelocity;
		PhaseUpperLin_MC_MoveAbsolute.Execute:=TRUE;
		fb_ton_debug_5.IN:=TRUE;
		PhaseUpperState:=2;
	2:
		IF NOT PhaseUpperLin_MC_MoveAbsolute.Done THEN
			PhaseUpperState:=2;
		ELSIF PhaseUpperLin_MC_MoveAbsolute.Done THEN
				PhaseUpperState:=88;
		END_IF
		IF PhaseUpperReset THEN
			PhaseUpperState:=89;
		END_IF

	88:
		PhaseUpperMove:=FALSE;
		PhaseUpperState:=0;
		PhaseUpperBusy:=FALSE;
		PhaseUpperDone:=TRUE;
		Error:=FALSE;
		ErrorID:=0;
		PhaseUpperLin_MC_MoveAbsolute.Execute:=FALSE;
		fb_ton_debug_5.IN:=FALSE;
	89:
		PhaseUpperMove:=FALSE;
		PhaseUpperState:=0;
		PhaseUpperBusy:=FALSE;
		PhaseUpperDone:=FALSE;
		Error:=FALSE;
		ErrorID:=0;
		PhaseUpperLin_MC_MoveAbsolute.Execute:=FALSE;
		fb_ton_debug_5.IN:=FALSE;
	99:
		PhaseUpperMove:=FALSE;
		PhaseUpperState:=99;
		PhaseUpperBusy:=FALSE;
		PhaseUpperDone:=FALSE;
		Error:=TRUE;
		PhaseUpperLin_MC_MoveAbsolute.Execute:=FALSE;
		fb_ton_debug_5.IN:=FALSE;
	-100:
		FB_PlcEmergencyStop();
		PhaseUpperMove:=FALSE;
		PhaseUpperState:=-100;
		PhaseUpperBusy:=FALSE;
		PhaseUpperDone:=FALSE;
		Error:=TRUE;
		PhaseUpperLin_MC_MoveAbsolute.Execute:=FALSE;
		fb_ton_debug_5.IN:=FALSE;
END_CASE
END_IF
END_ACTION

ACTION A_RightBottomMove:
IF RightBottomMove THEN
RightBottomBusy:=TRUE;
RightBottomDone:=FALSE;
fb_ton_debug_4(PT:=t#10s);
(*×îºóÔÙ¼ì²éÒ»±éñîºÏ£¬²»ñîºÏÎªÕýÈ·×´Ì¬*)
IF LeftTopLin.NcToPlc.CoupleState<>0 OR LeftBottomLin.NcToPlc.CoupleState<>0
			OR RightTopLin.NcToPlc.CoupleState<>0 OR RightBottomLin.NcToPlc.CoupleState<>0 THEN
			ErrorID:=1;
			RightBottomState:=-100;
END_IF
A_MoveMC();
CASE RightBottomState OF
	0:
		//IF Top_MC_MoveAbsolute.Error OR Bottom_MC_MoveAbsolute.Error
		//	OR RightTopLin_MC_MoveAbsolute.Error OR RightBottomLin_MC_MoveAbsolute.Error THEN		(*¼ì²éMC Error*)
		//	ErrorID:=2;
		//	RightBottomState:=99;
		IF leftTopLin.Status.NotMoving AND  leftBottomLin.Status.NotMoving
			 AND RightTopLin.Status.NotMoving AND RightBottomLin.Status.NotMoving THEN	(*Öá¶¼´¦ÓÚÍ£Ö¹×´Ì¬Ê±£¬×ªÏÂÒ»²½*)
			RightBottomState:=1;
		END_IF
	1:
		RightBottomLin_MC_MoveAbsolute.Position:=RightBottomPosition;
		RightBottomLin_MC_MoveAbsolute.Velocity:=RightBottomVelocity;
		RightBottomLin_MC_MoveAbsolute.Execute:=TRUE;
		fb_ton_debug_4.IN:=TRUE;
		RightBottomState:=2;
	2:
		IF LeftTopLin.Status.Moving OR RightTopLin.Status.Moving  OR LeftBottomLin.Status.Moving THEN	(*³ýÁËÔË¶¯Öá¶¯£¬ÆäÓàÖáÓÐ¶¯£¬´íÎó*)
			ErrorID:=3;
			RightBottomState:=-100;
		ELSIF NOT RightBottomLin_MC_MoveAbsolute.Done THEN		(*ÔË¶¯ÖÐ£¬¼ì²éDoneÐÅºÅ£¬Ã»ÓÐÔòÑ­»·£¬³¬Ê±±¨´í*)
			(*IF NOT  fb_ton.Q THEN
				LeftTopState:=2;
			ELSE
				ErrorID:=5;
				LeftTopState:=-100;
			END_IF*)
			RightBottomState:=2;
		ELSIF RightBottomLin_MC_MoveAbsolute.Done THEN		(*ÔË¶¯Íê³É£¬×ªÏÂÒ»²½*)
				RightBottomState:=88;
		END_IF
		(*½ÓÊÕµ½stopÐÅºÅÊ±£¬reset×´Ì¬*)
		IF RightBottomReset THEN
			RightBottomState:=89;
		END_IF

	88:
		RightBottomMove:=FALSE;
		RightBottomState:=0;
		RightBottomBusy:=FALSE;
		RightBottomDone:=TRUE;
		Error:=FALSE;
		ErrorID:=0;
		RightBottomLin_MC_MoveAbsolute.Execute:=FALSE;
		fb_ton_debug_4.IN:=FALSE;
	89:
		RightBottomMove:=FALSE;
		RightBottomState:=0;
		RightBottomBusy:=FALSE;
		RightBottomDone:=FALSE;
		Error:=FALSE;
		ErrorID:=0;
		RightBottomLin_MC_MoveAbsolute.Execute:=FALSE;
		fb_ton_debug_4.IN:=FALSE;
	99:
		RightBottomMove:=FALSE;
		RightBottomState:=99;
		RightBottomBusy:=FALSE;
		RightBottomDone:=FALSE;
		Error:=TRUE;
		RightBottomLin_MC_MoveAbsolute.Execute:=FALSE;
		fb_ton_debug_4.IN:=FALSE;
	-100:
		FB_PlcEmergencyStop();
		RightBottomMove:=FALSE;
		RightBottomState:=-100;
		RightBottomBusy:=FALSE;
		RightBottomDone:=FALSE;
		Error:=TRUE;
		RightBottomLin_MC_MoveAbsolute.Execute:=FALSE;
		fb_ton_debug_4.IN:=FALSE;
END_CASE
END_IF
END_ACTION

ACTION A_RightTopMove:
IF RightTopMove THEN
RightTopBusy:=TRUE;
RightTopDone:=FALSE;
fb_ton_debug_2(PT:=t#10s);
(*×îºóÔÙ¼ì²éÒ»±éñîºÏ£¬²»ñîºÏÎªÕýÈ·×´Ì¬*)
IF LeftTopLin.NcToPlc.CoupleState<>0 OR LeftBottomLin.NcToPlc.CoupleState<>0
			OR RightTopLin.NcToPlc.CoupleState<>0 OR RightBottomLin.NcToPlc.CoupleState<>0 THEN
			ErrorID:=1;
			RightTopState:=-100;
END_IF
A_MoveMC();
CASE RightTopState OF
	0:
		//IF Top_MC_MoveAbsolute.Error OR Bottom_MC_MoveAbsolute.Error
		//	OR RightTopLin_MC_MoveAbsolute.Error OR RightBottomLin_MC_MoveAbsolute.Error THEN		(*¼ì²éMC Error*)
		//	ErrorID:=2;
		//	RightTopState:=99;
		IF leftTopLin.Status.NotMoving AND  leftBottomLin.Status.NotMoving
			 AND RightTopLin.Status.NotMoving AND RightBottomLin.Status.NotMoving THEN	(*Öá¶¼´¦ÓÚÍ£Ö¹×´Ì¬Ê±£¬×ªÏÂÒ»²½*)
			RightTopState:=1;
		END_IF
	1:
		RightTopLin_MC_MoveAbsolute.Position:=RightTopPosition;
		RightTopLin_MC_MoveAbsolute.Velocity:=RightTopVelocity;
		RightTopLin_MC_MoveAbsolute.Execute:=TRUE;
		fb_ton_debug_2.IN:=TRUE;
		RightTopState:=2;
	2:
		IF LeftTopLin.Status.Moving OR LeftBottomLin.Status.Moving OR RightBottomLin.Status.Moving THEN	(*³ýÁËÔË¶¯Öá¶¯£¬ÆäÓàÖáÓÐ¶¯£¬´íÎó*)
			ErrorID:=3;
			RightTopState:=-100;
		ELSIF NOT RightTopLin_MC_MoveAbsolute.Done THEN		(*ÔË¶¯ÖÐ£¬¼ì²éDoneÐÅºÅ£¬Ã»ÓÐÔòÑ­»·£¬³¬Ê±±¨´í*)
			(*IF NOT  fb_ton.Q THEN
				LeftTopState:=2;
			ELSE
				ErrorID:=5;
				LeftTopState:=-100;
			END_IF*)
			RightTopState:=2;
		ELSIF RightTopLin_MC_MoveAbsolute.Done THEN		(*ÔË¶¯Íê³É£¬×ªÏÂÒ»²½*)
				RightTopState:=88;
		END_IF
		(*½ÓÊÕµ½stopÐÅºÅÊ±£¬reset×´Ì¬*)
		IF RightTopReset THEN
			RightTopState:=89;
		END_IF

	88:
		RightTopMove:=FALSE;
		RightTopState:=0;
		RightTopBusy:=FALSE;
		RightTopDone:=TRUE;
		Error:=FALSE;
		ErrorID:=0;
		RightTopLin_MC_MoveAbsolute.Execute:=FALSE;
		fb_ton_debug_2.IN:=FALSE;
	89:
		RightTopMove:=FALSE;
		RightTopState:=0;
		RightTopBusy:=FALSE;
		RightTopDone:=FALSE;
		Error:=FALSE;
		ErrorID:=0;
		RightTopLin_MC_MoveAbsolute.Execute:=FALSE;
		fb_ton_debug_2.IN:=FALSE;
	99:
		RightTopMove:=FALSE;
		RightTopState:=99;
		RightTopBusy:=FALSE;
		RightTopDone:=FALSE;
		Error:=TRUE;
		RightTopLin_MC_MoveAbsolute.Execute:=FALSE;
		fb_ton_debug_2.IN:=FALSE;
	-100:
		FB_PlcEmergencyStop();
		RightTopMove:=FALSE;
		RightTopState:=-100;
		RightTopBusy:=FALSE;
		RightTopDone:=FALSE;
		Error:=TRUE;
		RightTopLin_MC_MoveAbsolute.Execute:=FALSE;
		fb_ton_debug_2.IN:=FALSE;
END_CASE
END_IF
END_ACTION

ACTION A_TaperMove:
IF TaperMove THEN
TaperBusy:=TRUE;
TaperDone:=FALSE;
fb_ton(PT:=t#80s);
(*×îºóÔÙ¼ì²éÒ»±éñîºÏ£¬²»ñîºÏÎªÕýÈ·×´Ì¬*)
IF LeftTopLin.NcToPlc.CoupleState<>0 OR LeftBottomLin.NcToPlc.CoupleState<>0
			OR RightTopLin.NcToPlc.CoupleState<>0 OR RightBottomLin.NcToPlc.CoupleState<>0 THEN
			ErrorID:=1;
			TaperState:=-100;
END_IF
(*×ó²àÉÏÏÂÖá¶¯£¬ESTOP*)
IF LeftTopLin.Status.Moving OR LeftBottomLin.Status.Moving THEN
			ErrorID:=2;
			TaperState:=-100;
END_IF
(*ÓÒÉÏ¶¯¡¢ÓÒÏÂ²»¶¯£¬»òÕßÓÒÏÂ¶¯¡¢ÓÒÉÏ²»¶¯¡£ESTOP*)
IF (RightTopLin.Status.Moving AND RightBottomLin.Status.NotMoving) OR (RightTopLin.Status.NotMoving AND RightBottomLin.Status.Moving) THEN
			ErrorID:=3;
			TaperState:=-100;
END_IF
A_MoveMC();
CASE TaperState OF

	0:
		IF RightTopLin.Status.Moving OR RightBottomLin.Status.Moving THEN	(*ÓÒ²àÉÏÏÂÖáÕýÔÚÔËÐÐ£¬Ñ­»·¸Ã²½µÈ´ý*)
			TaperState:=88;
		ELSIF Top_MC_MoveAbsolute.Error OR Bottom_MC_MoveAbsolute.Error THEN		(*¼ì²éMC Error*)
			ErrorID:=4;
			TaperState:=99;
		ELSIF leftTopLin.Status.NotMoving AND  leftBottomLin.Status.NotMoving
			 AND RightTopLin.Status.NotMoving AND RightBottomLin.Status.NotMoving THEN	(*Öá¶¼´¦ÓÚÍ£Ö¹×´Ì¬Ê±£¬×ªÏÂÒ»²½*)
			TaperState:=1;
		END_IF
	1:
		RightTopLin_MC_MoveAbsolute.Position:=TaperPosition;
		RightTopLin_MC_MoveAbsolute.Velocity:=TaperVelocity;
		RightBottomLin_MC_MoveAbsolute.Position:=TaperPosition;
		RightBottomLin_MC_MoveAbsolute.Velocity:=TaperVelocity;
		RightTopLin_MC_MoveAbsolute.Execute:=TRUE;
		RightBottomLin_MC_MoveAbsolute.Execute:=TRUE;
		fb_ton.IN:=TRUE;
		TaperState:=2;
	2:
		IF leftTopLin.Status.Moving OR   leftBottomLin.Status.Moving THEN		(*×ó²àÉÏÏÂÖá¶¯£¬ESTOP*)
			ErrorID:=5;
			TaperState:=-100;
		ELSIF  (RightTopLin.Status.Moving AND RightBottomLin.Status.NotMoving) OR (RightTopLin.Status.NotMoving AND RightBottomLin.Status.Moving) THEN
			ErrorID:=6;
			TaperState:=-100;
		ELSIF NOT RightTopLin_MC_MoveAbsolute.Done OR NOT  RightBottomLin_MC_MoveAbsolute.Done THEN		(*ÔË¶¯ÖÐ£¬¼ì²éDoneÐÅºÅ£¬Ã»ÓÐÔòÑ­»·£¬³¬Ê±±¨´í*)
			(*IF NOT  fb_ton.Q THEN
				TaperState:=2;
			ELSE
				ErrorID:=5;
				TaperState:=-100;
			END_IF*)
			TaperState:=2;
		ELSIF RightTopLin_MC_MoveAbsolute.Done  AND  RightBottomLin_MC_MoveAbsolute.Done THEN		(*ÔË¶¯Íê³É£¬×ªÏÂÒ»²½*)
				TaperState:=88;
		END_IF
		(*½ÓÊÕµ½stopÐÅºÅÊ±£¬reset×´Ì¬*)
		IF TaperReset THEN
			TaperState:=89;
		END_IF

	88:
		TaperMove:=FALSE;
		TaperState:=0;
		TaperBusy:=FALSE;
		TaperDone:=TRUE;
		Error:=FALSE;
		ErrorID:=0;
		RightTopLin_MC_MoveAbsolute.Execute:=FALSE;
		RightBottomLin_MC_MoveAbsolute.Execute:=FALSE;
		fb_ton.IN:=FALSE;
	89:
		TaperMove:=FALSE;
		TaperState:=0;
		TaperBusy:=FALSE;
		TaperDone:=FALSE;
		Error:=FALSE;
		ErrorID:=0;
		RightTopLin_MC_MoveAbsolute.Execute:=FALSE;
		RightBottomLin_MC_MoveAbsolute.Execute:=FALSE;
		fb_ton.IN:=FALSE;
	99:
		TaperMove:=FALSE;
		TaperState:=99;
		TaperBusy:=FALSE;
		TaperDone:=FALSE;
		Error:=TRUE;
		RightTopLin_MC_MoveAbsolute.Execute:=FALSE;
		RightBottomLin_MC_MoveAbsolute.Execute:=FALSE;
		fb_ton.IN:=FALSE;
	-100:
		FB_PlcEmergencyStop();
		TaperMove:=FALSE;
		TaperState:=-100;
		TaperBusy:=FALSE;
		TaperDone:=FALSE;
		Error:=TRUE;
		RightTopLin_MC_MoveAbsolute.Execute:=FALSE;
		RightBottomLin_MC_MoveAbsolute.Execute:=FALSE;
		fb_ton.IN:=FALSE;
END_CASE
END_IF
END_ACTION

ACTION A_TopMove:
IF TopMove THEN
TopBusy:=TRUE;
TopDone:=FALSE;
fb_ton1(PT:=t#80s);(*2mm/s max spees,120mmÐÐ³Ì£¬60sÄÚ×ßÍê*)
A_MoveMC();
CASE TopState OF
	0:
		//IF Top_MC_MoveAbsolute.Error OR RightTopLin_MC_MoveAbsolute.Error THEN		(*¼ì²éMC Error*)
		//	ErrorID:=2;
		//	TopState:=99;
		//END_IF
		TopState:=1;
	1:
		Top_MC_MoveAbsolute.Position:=TopPosition;
		Top_MC_MoveAbsolute.Velocity:=TopVelocity;
		Top_MC_MoveAbsolute.Execute:=TRUE;
		RightTopLin_MC_MoveAbsolute.Position:=TopPosition;
		RightTopLin_MC_MoveAbsolute.Velocity:=TopVelocity;
		RightTopLin_MC_MoveAbsolute.Execute:=TRUE;
		fb_ton1.IN:=TRUE;
		TopState:=2;
	2:
		IF leftBottomLin.Status.Moving OR RightBottomLin.Status.Moving THEN	(*ÏÂÁº¶¯,ESTOP*)
			ErrorID:=3;
			TopState:=-100;
		ELSIF  (LeftTopLin.Status.Moving AND  RightTopLin.Status.NotMoving)
				OR (RightTopLin.Status.Moving AND  LeftTopLin.Status.NotMoving) THEN			(*Ò»Öá¶¯£¬ÁíÒ»Öá²»¶¯£¬½ô¼±×´Ì¬*)
			//ErrorID:=4;
			//TopState:=-100;
		ELSIF NOT Top_MC_MoveAbsolute.Done OR NOT RightTopLin_MC_MoveAbsolute.Done THEN		(*ÔË¶¯ÖÐ£¬¼ì²éDoneÐÅºÅ£¬Ã»ÓÐÔòÑ­»·£¬³¬Ê±±¨´í*)
			TopState:=2;
		ELSIF Top_MC_MoveAbsolute.Done AND RightTopLin_MC_MoveAbsolute.Done THEN		(*ÔË¶¯Íê³É£¬×ªÏÂÒ»²½*)
				TopState:=88;
		END_IF
		(*½ÓÊÕµ½stopÐÅºÅÊ±£¬reset×´Ì¬*)
		IF TopReset THEN
			TopState:=89;
		END_IF

	88:
		TopMove:=FALSE;
		TopState:=0;
		TopBusy:=FALSE;
		TopDone:=TRUE;
		Error:=FALSE;
		ErrorID:=0;
		Top_MC_MoveAbsolute.Execute:=FALSE;
		RightTopLin_MC_MoveAbsolute.Execute:=FALSE;
		fb_ton1.IN:=FALSE;
	89:
		TopMove:=FALSE;
		TopState:=0;
		TopBusy:=FALSE;
		TopDone:=FALSE;
		Error:=FALSE;
		ErrorID:=0;
		Top_MC_MoveAbsolute.Execute:=FALSE;
		RightTopLin_MC_MoveAbsolute.Execute:=FALSE;
		fb_ton1.IN:=FALSE;
	99:
		TopMove:=FALSE;
		TopState:=99;
		TopBusy:=FALSE;
		TopDone:=FALSE;
		Error:=TRUE;
		Top_MC_MoveAbsolute.Execute:=FALSE;
		RightTopLin_MC_MoveAbsolute.Execute:=FALSE;
		fb_ton1.IN:=FALSE;
	-100:
		FB_PlcEmergencyStop();
		TopMove:=FALSE;
		TopState:=-100;
		TopBusy:=FALSE;
		TopDone:=FALSE;
		Error:=TRUE;
		Top_MC_MoveAbsolute.Execute:=FALSE;
		RightTopLin_MC_MoveAbsolute.Execute:=FALSE;
		fb_ton1.IN:=FALSE;
END_CASE
END_IF
END_ACTION

END_FUNCTION_BLOCK

(* stored: Version 1.1.0.1, ProductVersion 3.1.4024.6
   POU FB_Move: Id {f9a99ade-b4af-4565-bffe-bba1640e411e}, SpecialFunc None
   Action A_BCGapMove: Id {14a23b8d-1d11-4027-a881-ef621e956d3f}
   Action A_BCGapMove_2: Id {515559be-7182-4ea3-a18e-2b792ce3b070}
   Action A_BottomMove: Id {b44a7ecd-72fc-446a-9274-88916c5022c8}
   Action A_GapMove: Id {ea782744-09ee-4428-bf59-993d9a34c853}
   Action A_LeftBottomMove: Id {435e4286-c6ed-406e-a3b9-a54ace766d6c}
   Action A_LeftTopMove: Id {c3c5ae62-8709-476f-aa75-1e25179f7e02}
   Action A_MoveMC: Id {f577884c-c19e-4448-8f5c-62de64b66e2f}
   Action A_PhaseLowerMove: Id {b176c8c4-3648-4101-9537-ebcaf72117e6}
   Action A_PhaseUpperMove: Id {c71114c4-8dd7-4dff-a0c8-2b16b3228dc3}
   Action A_RightBottomMove: Id {18336067-1624-4437-bf3d-756ffa42f33f}
   Action A_RightTopMove: Id {74383921-9bde-4a33-845f-0695282e023f}
   Action A_TaperMove: Id {4bc4b766-d1e2-45d6-844f-b936dd8e4ded}
   Action A_TopMove: Id {d95f110f-5f71-4103-b00f-7eb6334d6024} *)
